# EPICS StreamDevice protocol: motorseqIOC/protocols/motorProto.proto
OutTerminator = CR;
InTerminator = CR LF;

move_relative{
	out "%(\$1)iPR%i";
}
